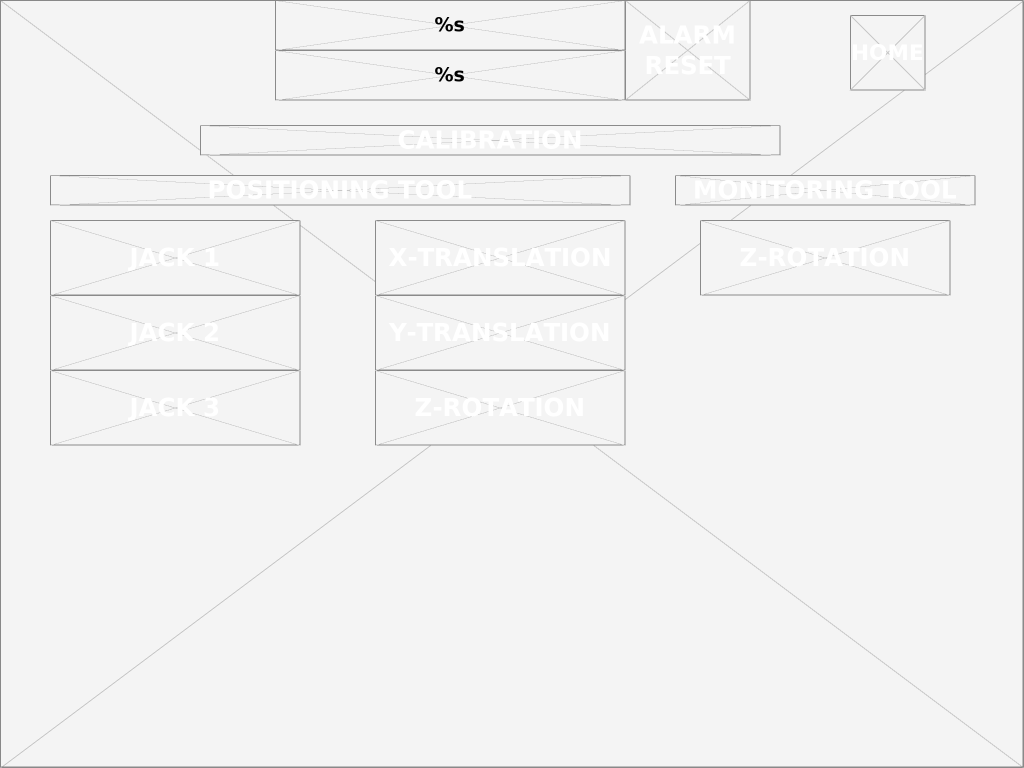
VISUALIZATION CALIBRATION_SCREEN  // 1024x768
    Image (0,0 1024x768), image: ImagePool.background1
    Image (50,220 250x75), "JACK 1", image: ImagePool.PB_BU_250_75
        OnMouseDown: execute { MAIN.Visualization.P12B_Calibrate_Jack1.Active := TRUE; }
        OnMouseUp: execute { MAIN.Visualization.P12B_Calibrate_Jack1.Active := FALSE; }
    Image (50,370 250x75), "JACK 3", image: ImagePool.PB_BU_250_75
        OnMouseDown: execute { MAIN.Visualization.P12B_Calibrate_Jack3.Active := TRUE; }
        OnMouseUp: execute { MAIN.Visualization.P12B_Calibrate_Jack2.Active := FALSE; }
    Image (50,295 250x75), "JACK 2", image: ImagePool.PB_BU_250_75
        OnMouseDown: execute { MAIN.Visualization.P12B_Calibrate_Jack2.Active := TRUE; }
        OnMouseUp: execute { MAIN.Visualization.P12B_Calibrate_Jack2.Active := FALSE; }
    Image (375,370 250x75), "Z-ROTATION", image: ImagePool.PB_BU_250_75
        OnMouseDown: execute { MAIN.Visualization.P12B_Calibrate_PosTool_RotZ.Active := TRUE; }
        OnMouseUp: execute { MAIN.Visualization.P12B_Calibrate_PosTool_RotZ.Active := FALSE; }
    Image (700,220 250x75), "Z-ROTATION", image: ImagePool.PB_BU_250_75
        OnMouseDown: execute { MAIN.Visualization.P12B_Calibrate_MonTool_RotZ.Active := TRUE; }
        OnMouseUp: execute { MAIN.Visualization.P12B_Calibrate_MonTool_RotZ.Active := FALSE; }
    Image (625,0 125x100), "ALARM RESET", image: ImagePool.PB_BU_125_100
        p84334746: MAIN.Visualization.P00B_Alarm_Reset.bitmap_ID
        OnMouseDown: execute { MAIN.Visualization.P00B_Alarm_Reset.Active:=TRUE; }
        OnMouseUp: execute { MAIN.Visualization.P00B_Alarm_Reset.Active:=FALSE; }
    Image (275,0 350x50), "%s", text variable: MAIN.Visualization.P00D_Station_Status.display_text, image: ImagePool.IN_BU_300_50
        p84334746: MAIN.Visualization.P00D_Station_Status.bitmap_ID
    Image (275,50 350x50), "%s", text variable: MAIN.Visualization.P00D_Alarm_Status.display_text, image: ImagePool.IN_BU_300_50
        p84334746: MAIN.Visualization.P00D_Alarm_Status.bitmap_ID
    Image (200,125 580x30), "CALIBRATION", image: VisuDialogs.ImagePoolDialogs.Title2
    Image (50,175 580x30), "POSITIONING TOOL", image: VisuDialogs.ImagePoolDialogs.Title2
    Image (675,175 300x30), "MONITORING TOOL", image: VisuDialogs.ImagePoolDialogs.Title
    Image (375,295 250x75), "Y-TRANSLATION", image: ImagePool.PB_BU_250_75
        OnMouseDown: execute { MAIN.Visualization.P12B_Calibrate_YTRANS.Active := TRUE; }
        OnMouseUp: execute { MAIN.Visualization.P12B_Calibrate_YTRANS.Active := FALSE; }
    Image (375,220 250x75), "X-TRANSLATION", image: ImagePool.PB_BU_250_75
        OnMouseDown: execute { MAIN.Visualization.P12B_Calibrate_XTRANS.Active := TRUE; }
        OnMouseUp: execute { MAIN.Visualization.P12B_Calibrate_XTRANS.Active := FALSE; }
    Image (850,15 75x75), "HOME", image: ImagePool.PB_BU_75_75
        OnMouseDown: execute { MAIN.Visualization.P12B_HOME_SCREEN.Active := TRUE; }
        OnMouseUp: execute { MAIN.Visualization.P12B_HOME_SCREEN.Active := FALSE; }
END_VISUALIZATION

(* stored: Version 1.1.0.1, ProductVersion 3.1.4024.0
   Visu CALIBRATION_SCREEN: Id {3b2de891-9433-418a-b93a-f89799353c28} *)
